# EPICS autosave request: apps/omegaCYD218App/Db/OmegaCYD218_chN_settings.req
#
# Omega CYD218 Series Digital Thermometers
#
$(P)$(CH)desc
$(P)$(CH)inputSet
$(P)$(CH)curveSet
